(* IEC 61131-3 sources: stc/testdata/parse, 2 files *)

(* ---- motor_control.st ---- *)
FUNCTION_BLOCK FB_Motor
VAR_INPUT
    Start : BOOL;
    Stop  : BOOL;
END_VAR
VAR_OUTPUT
    Running : BOOL;
END_VAR
IF Start AND NOT Stop THEN
    Running := TRUE;
ELSIF Stop THEN
    Running := FALSE;
END_IF;
END_FUNCTION_BLOCK

(* ---- broken_input.st ---- *)
PROGRAM Broken
VAR
    x : BOOL
END_VAR
IF x THEN
    y := ;
END_IF;
x := TRUE;
END_PROGRAM
